// This interface represents a logger for error messages.
INTERFACE I_ErrorLogger EXTENDS __SYSTEM.IQueryInterface

// Logs the provided error message.
METHOD Invoke
VAR_INPUT
	ipError : I_Error;	 // The error message to be logged.
END_VAR
VAR_OUTPUT
	bIsBusy : BOOL;		// Is the operation still executing?
	Error 	: T_Error;	// Error produced by operation.
END_VAR
END_METHOD

END_INTERFACE

(* stored: Version 1.1.0.1
   Itf I_ErrorLogger: Id {2a6c0c04-196a-0850-13cc-02c2e4d81abb}
   Method Invoke: Id {fe10df30-9b43-0b6f-3ff3-133dc5932ce3} *)
